// Mitsubishi GX Works2 project: StationMovement   PLC: Q02U

PROGRAM MAIN
VAR
  Station_1 : Station;
  control_2 : control;
END_VAR
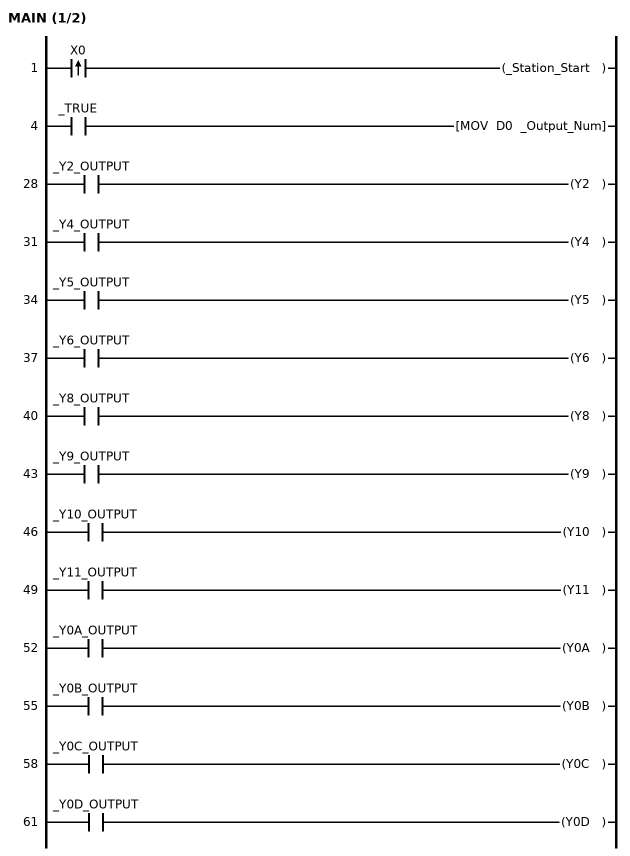
; FB BLK START Station(Station_1)
1     LDP     X0
      OUT     _Station_Start
4     LD      _TRUE
      MOV     D0 _Output_Num
; FB START
; FB_NAME Station
; INSTANCE_NAME Station_1
; FB IN_B:Station_Start
; FB OUT_Y2_OUTPUT:B
; FB IN_W:Output_Num
; FB OUT_Y4_OUTPUT:B
; FB OUT_Y5_OUTPUT:B
; FB OUT_Y6_OUTPUT:B
; FB OUT_Y8_OUTPUT:B
; FB OUT_Y9_OUTPUT:B
; FB OUT_Y10_OUTPUT:B
; FB OUT_Y11_OUTPUT:B
; FB OUT_Y0A_OUTPUT:B
; FB OUT_Y0B_OUTPUT:B
; FB OUT_Y0C_OUTPUT:B
; FB OUT_Y0D_OUTPUT:B
; FB OUT_Num:W
; FB END
28    LD      _Y2_OUTPUT
      OUT     Y2
31    LD      _Y4_OUTPUT
      OUT     Y4
34    LD      _Y5_OUTPUT
      OUT     Y5
37    LD      _Y6_OUTPUT
      OUT     Y6
40    LD      _Y8_OUTPUT
      OUT     Y8
43    LD      _Y9_OUTPUT
      OUT     Y9
46    LD      _Y10_OUTPUT
      OUT     Y10
49    LD      _Y11_OUTPUT
      OUT     Y11
52    LD      _Y0A_OUTPUT
      OUT     Y0A
55    LD      _Y0B_OUTPUT
      OUT     Y0B
58    LD      _Y0C_OUTPUT
      OUT     Y0C
61    LD      _Y0D_OUTPUT
      OUT     Y0D
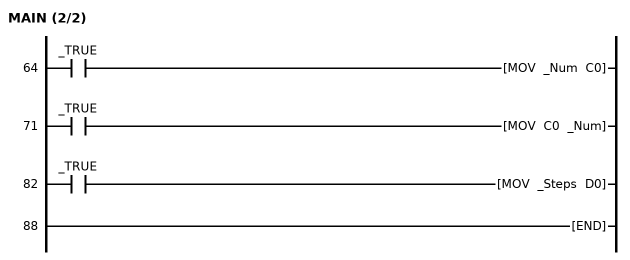
64    LD      _TRUE
      MOV     _Num C0
; FB BLK END
; FB BLK START control(control_2)
71    LD      _TRUE
      MOV     C0 _Num
; FB START
; FB_NAME control
; INSTANCE_NAME control_2
; FB IN_W:Num
; FB OUT_Steps:W
; FB END
82    LD      _TRUE
      MOV     _Steps D0
; FB BLK END
88    END
END_PROGRAM

FUNCTION_BLOCK Station
VAR_INPUT
  Station_Start : BOOL;
END_VAR
VAR_OUTPUT
  Y2_OUTPUT : BOOL;
  Y4_OUTPUT : BOOL;
  Y5_OUTPUT : BOOL;
  Y6_OUTPUT : BOOL;
  Y8_OUTPUT : BOOL;
  Y9_OUTPUT : BOOL;
  Y10_OUTPUT : BOOL;
  Y11_OUTPUT : BOOL;
  Y0A_OUTPUT : BOOL;
  Y0B_OUTPUT : BOOL;
END_VAR
VAR_INPUT
  Output_Num : INT;
END_VAR
VAR_OUTPUT
  Num : INT;
  Y0C_OUTPUT : BOOL;
  Y0D_OUTPUT : BOOL;
END_VAR
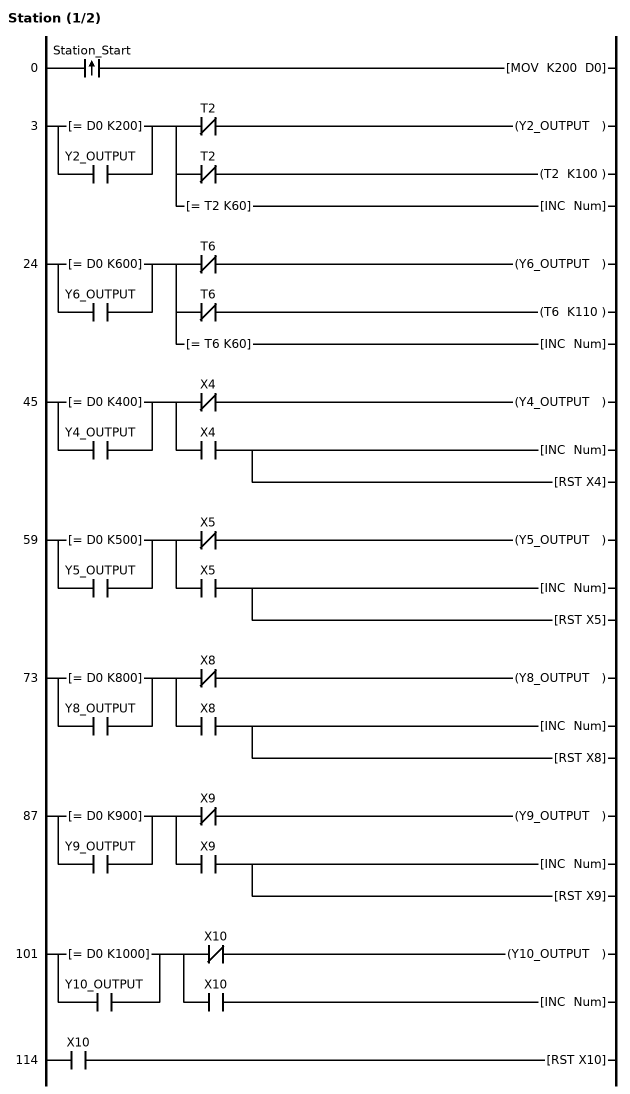
0     LDP     Station_Start
      MOV     K200 D0
3     LD=     D0 K200
      OR      Y2_OUTPUT
      MPS
      ANI     T2
      OUT     Y2_OUTPUT
      MRD
      ANI     T2
      OUT     T2 K100
      MPP
      AND=    T2 K60
      INC     Num
24    LD=     D0 K600
      OR      Y6_OUTPUT
      MPS
      ANI     T6
      OUT     Y6_OUTPUT
      MRD
      ANI     T6
      OUT     T6 K110
      MPP
      AND=    T6 K60
      INC     Num
45    LD=     D0 K400
      OR      Y4_OUTPUT
      MPS
      ANI     X4
      OUT     Y4_OUTPUT
      MPP
      AND     X4
      INC     Num
      RST     X4
59    LD=     D0 K500
      OR      Y5_OUTPUT
      MPS
      ANI     X5
      OUT     Y5_OUTPUT
      MPP
      AND     X5
      INC     Num
      RST     X5
73    LD=     D0 K800
      OR      Y8_OUTPUT
      MPS
      ANI     X8
      OUT     Y8_OUTPUT
      MPP
      AND     X8
      INC     Num
      RST     X8
87    LD=     D0 K900
      OR      Y9_OUTPUT
      MPS
      ANI     X9
      OUT     Y9_OUTPUT
      MPP
      AND     X9
      INC     Num
      RST     X9
101   LD=     D0 K1000
      OR      Y10_OUTPUT
      MPS
      ANI     X10
      OUT     Y10_OUTPUT
      MPP
      AND     X10
      INC     Num
114   LD      X10
      RST     X10
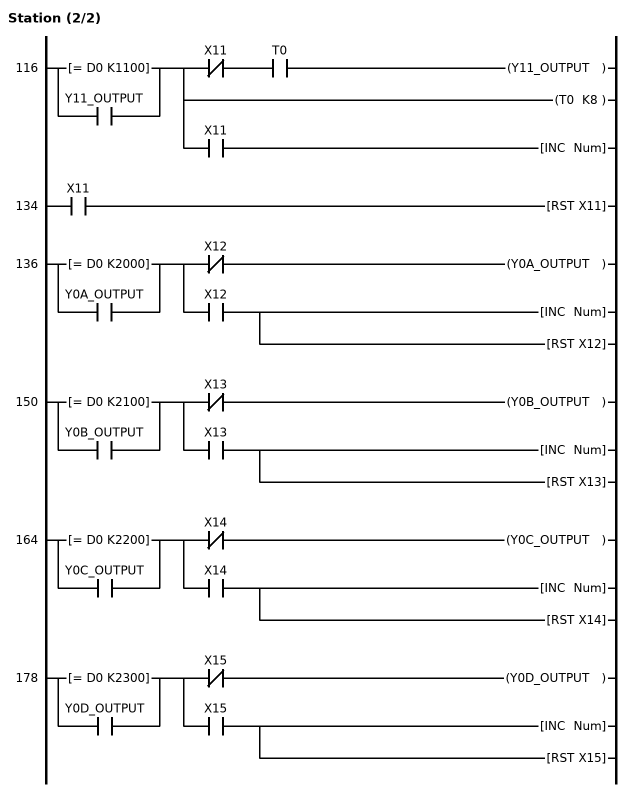
116   LD=     D0 K1100
      OR      Y11_OUTPUT
      MPS
      ANI     X11
      AND     T0
      OUT     Y11_OUTPUT
      MPP
      OUT     T0 K8
      AND     X11
      INC     Num
134   LD      X11
      RST     X11
136   LD=     D0 K2000
      OR      Y0A_OUTPUT
      MPS
      ANI     X12
      OUT     Y0A_OUTPUT
      MPP
      AND     X12
      INC     Num
      RST     X12
150   LD=     D0 K2100
      OR      Y0B_OUTPUT
      MPS
      ANI     X13
      OUT     Y0B_OUTPUT
      MPP
      AND     X13
      INC     Num
      RST     X13
164   LD=     D0 K2200
      OR      Y0C_OUTPUT
      MPS
      ANI     X14
      OUT     Y0C_OUTPUT
      MPP
      AND     X14
      INC     Num
      RST     X14
178   LD=     D0 K2300
      OR      Y0D_OUTPUT
      MPS
      ANI     X15
      OUT     Y0D_OUTPUT
      MPP
      AND     X15
      INC     Num
      RST     X15
END_FUNCTION_BLOCK

FUNCTION_BLOCK control
VAR_INPUT
  Num : INT;
END_VAR
VAR_OUTPUT
  Steps : INT;
END_VAR
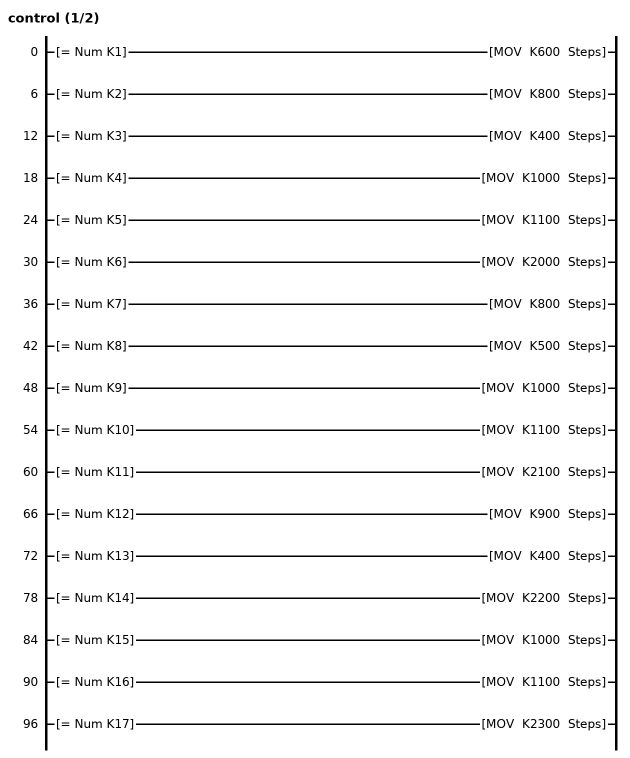
0     LD=     Num K1
      MOV     K600 Steps
6     LD=     Num K2
      MOV     K800 Steps
12    LD=     Num K3
      MOV     K400 Steps
18    LD=     Num K4
      MOV     K1000 Steps
24    LD=     Num K5
      MOV     K1100 Steps
30    LD=     Num K6
      MOV     K2000 Steps
36    LD=     Num K7
      MOV     K800 Steps
42    LD=     Num K8
      MOV     K500 Steps
48    LD=     Num K9
      MOV     K1000 Steps
54    LD=     Num K10
      MOV     K1100 Steps
60    LD=     Num K11
      MOV     K2100 Steps
66    LD=     Num K12
      MOV     K900 Steps
72    LD=     Num K13
      MOV     K400 Steps
78    LD=     Num K14
      MOV     K2200 Steps
84    LD=     Num K15
      MOV     K1000 Steps
90    LD=     Num K16
      MOV     K1100 Steps
96    LD=     Num K17
      MOV     K2300 Steps
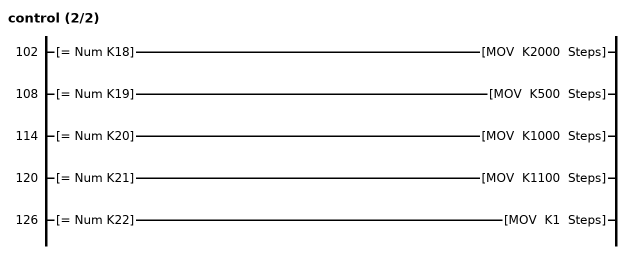
102   LD=     Num K18
      MOV     K2000 Steps
108   LD=     Num K19
      MOV     K500 Steps
114   LD=     Num K20
      MOV     K1000 Steps
120   LD=     Num K21
      MOV     K1100 Steps
126   LD=     Num K22
      MOV     K1 Steps
END_FUNCTION_BLOCK
